FUNCTION_BLOCK AllOtherDls
VAR
	OneDI: Lib.OneDI;
	PSU1 	AT %I* : BOOL;
	PSU2 	AT %I* : BOOL;
	FAP_PNL AT %I* : BOOL;
	FAP_LOOP_ALM AT %I* : BOOL;
	Telce_ASD_A_PNL_ALM AT %I* : BOOL;
	


END_VAR

END_FUNCTION_BLOCK

(* stored: Version 1.1.0.1, ProductVersion 3.1.4024.12
   POU AllOtherDls: Id {07162dc3-8969-46a4-a91e-5d7a6e5b8bcb}, SpecialFunc None *)
